// TIA Portal V16 export
// export: Created 2022-03-28T07:44:07.7346109Z, ExportSetting WithDefaults, DisplayName Totally Integrated Automation Portal, DisplayVersion V16 Update 5, DisplayName TIA Portal Version Control Interface, DisplayVersion V16 Update 2, DisplayName TIA Portal Openness, DisplayVersion V16 Update 5, DisplayName STEP 7 Professional, DisplayVersion V16 Update 5, DisplayName STEP 7 Safety, DisplayVersion V16, DisplayName WinCC Professional, DisplayVersion V16 Update 5
DATA_BLOCK "db_HMI"   // DB100
{ S7_Optimized_Access := 'FALSE' }
VERSION : 0.1
// stored: AutoNumber false, IsOnlyStoredInLoadMemory false, IsWriteProtectedInAS false
   VAR
      ariScreen : Array[0..3] of Int;
      iScreenNumbver : Int;
      bLights : Bool;
      bResetCycleKey : Bool;
      diPartsCounter : DInt;
      iPart_1 : Int;
      iPart_2 : Int;
      iPart_3 : Int;
      iPart_4 : Int;
      iPart_5 : Int;
      iPart_6 : Int;
      iPart_7 : Int;
      iPart_8 : Int;
      iPart_9 : Int;
      iPart_10 : Int;
   END_VAR
BEGIN
END_DATA_BLOCK
